(*********************************** G.D S.p.A. - Technical Department ***********************************
============= PROGRAM INFO ============
FOLDER:             TBD
MACHINES INVOLVED:  TBD 

============= DESCRIPTION =============
csp machine safety interfaces definition

============= REVISIONS ===============
Date		Version	 	Author      	Description             
----------	-------		------------  	--------------------------------------------
2019/04/24 	0000.00	 	M.Grasso		Creation of the PRG

**********************************************************************************************************)
(*$R
	process_ref := prc;
$*)
PROGRAM csp_main_safety_interface
VAR
	prc:						process;
	prc_path:					STRING;
		
END_VAR

_read_var_input();

_object_manager();

IF NOT objects_running()
THEN
	RETURN;	
END_IF

_read_process_image();

_mode_manager();

CASE process_get_mode(prc) of
	MODE_ABSENT,
	MODE_INACTIVE:
		RETURN;
	MODE_TEST:
		_handle_process_test();
END_CASE

_set_runtime_properties();

(********************************* BODY *********************************)

(************************************************************************)

_handle_messages();

_write_output();

ACTION _handle_messages:
;
END_ACTION

ACTION _handle_process_test:
;
END_ACTION

ACTION _mode_manager:
IF process_mode_req_is_pending(prc)
THEN
    process_apply_mode_req_first_step(prc);
    CASE process_get_mode(prc) OF
        MODE_TO_ABSENT:
			;
        MODE_TO_INACTIVE:
			;
        MODE_TO_TEST:
			;
        MODE_TO_OPERATIONAL:
			;
    END_CASE
    process_apply_mode_req_second_step(prc);
END_IF
END_ACTION

ACTION _object_manager:
IF objects_initialization()
THEN
	sub_process_init(
		object_name								:= 'csp_main_safety_interface.prc', 
		process									:= csp_main_safety.prc, 
		CONVERSION_this							:= prc);
		
	prc_path 									:= process_get_path(prc);
	
END_IF

IF objects_running()
THEN
	process_cycle(prc);
END_IF
END_ACTION

ACTION _read_process_image:
;
END_ACTION

ACTION _read_var_input:
;
END_ACTION

ACTION _set_runtime_properties:
;
END_ACTION

ACTION _write_output:
;
END_ACTION

END_PROGRAM

(* stored: Version 1.1.0.1, ProductVersion 3.1.4022.12
   POU csp_main_safety_interface: Id {accaf545-6a8a-4c1b-8746-1d8a689547bc}, SpecialFunc None
   Action _handle_messages: Id {13277fd1-f16d-435f-a47f-7829ca52ff7b}
   Action _handle_process_test: Id {abbba029-381a-4e61-a3f9-3adcde822894}
   Action _mode_manager: Id {29302d30-98e0-42fe-a14b-1579c802fe6f}
   Action _object_manager: Id {3ba29f0e-ad14-49b2-bf16-37e951a942fd}
   Action _read_process_image: Id {44cd3c4a-e4cc-4ccb-97c1-0dcd0a9a9488}
   Action _read_var_input: Id {b3882761-f046-4fdb-92cd-73bb08192f83}
   Action _set_runtime_properties: Id {6f4509bb-3387-4989-acb8-d2945d6fe20a}
   Action _write_output: Id {1cd61d08-1dee-4686-ad9f-004882d81e6d} *)
